// TIA Portal V20 export
FUNCTION_BLOCK "FB_Axis"   // FB410, SCL
{ S7_Optimized_Access := 'TRUE' }
// stored: AutoNumber false, MemoryReserve 100, SetENOAutomatically false
   VAR
      "sBrakeTest ZM" { S7_SetPoint := 'True'} : "FB_BrakeTest";
      "sBrakeTest ZL" { S7_SetPoint := 'True'} : "FB_BrakeTest";
      "BrakeTest ZM" : Struct
         sSBTDone { S7_SetPoint := 'True'} : Bool;
         sStartSBT { S7_SetPoint := 'True'} : Bool;
         sDone { S7_SetPoint := 'True'} : Bool;
         sError : Bool;
         sStateNum : Int;
         sDiagnoseError : Int;
         scloseExternalBrake : Bool;
      END_STRUCT;
      "BrakeTest ZL" : Struct
         sSBTDone { S7_SetPoint := 'True'} : Bool;
         sStartSBT { S7_SetPoint := 'True'} : Bool;
         sDone { S7_SetPoint := 'True'} : Bool;
         sError : Bool;
         sStateNum : Int;
         sDiagnoseError : Int;
         scloseExternalBrake : Bool;
      END_STRUCT;
      sErrorN : Array[1..8] of Bool;
      sTestStopRequested : Bool;
      sTestStopStart : Bool;
      sTestStopError : Bool;
      sTestStopEnd : Bool;
      sTestStopDone : Bool;
      sLedSITestOK : Bool;
      sLedSITestSlowFlashing : Bool;
      sLedSITestQuickFlashing : Bool;
      sTimerTestStopStart : TON_TIME;
      sTimerTestStopEnd : TON_TIME;
   END_VAR
   VAR RETAIN
      DisableAxis01_X { S7_SetPoint := 'True'} : Bool;
      DisableAxis02_Y { S7_SetPoint := 'True'} : Bool;
      DisableAxis03_ZM { S7_SetPoint := 'True'} : Bool;
      DisableAxis04_B { S7_SetPoint := 'True'} : Bool;
      DisableAxis05_U1 { S7_SetPoint := 'True'} : Bool;
      DisableAxis06_U2 { S7_SetPoint := 'True'} : Bool;
      DisableAxis07_V { S7_SetPoint := 'True'} : Bool;
      DisableAxis08_W { S7_SetPoint := 'True'} : Bool;
      DisableAxis09_ZL { S7_SetPoint := 'True'} : Bool;
   END_VAR
BEGIN
   REGION Description header 
       //==================================================================================
       // POSALUX Swiss SA / (C) Copyright 2025
       //----------------------------------------------------------------------------------
       // Title: FB_Axis
       // Comment/Function: 
       // Author: Fabien WALDT
       // Engineering: TIA Portal v17
       //----------------------------------------------------------------------------------
       // Change log table:
       // Version  | Date     | Expert in charge | Changes applied
       // ---------|----------|------------------|-----------------------------------------
       // 00.00.01 | 20250423 | WFA              | First released version
       // =================================================================================
   END_REGION

   REGION Axis disable
       "LBP_Axis01_X".A_ASpDisable  := FALSE;
       "LBP_Axis02_Y".A_ASpDisable  := FALSE;
       "LBP_Axis03_ZM".A_ASpDisable := FALSE;
       "LBP_Axis04_B".A_ASpDisable  := FALSE;
       "LBP_Axis05_U1".A_ASpDisable := FALSE;
       "LBP_Axis06_U2".A_ASpDisable := FALSE;
       "LBP_Axis07_V".A_ASpDisable  := FALSE;
       "LBP_Axis08_W".A_ASpDisable  := FALSE;
       "LBP_Axis09_ZL".A_ASpDisable := FALSE;
   END_REGION

   REGION Axis follow-up mode
       "LBP_Axis01_X".A_Follow_upMode  := TRUE;
       "LBP_Axis02_Y".A_Follow_upMode  := TRUE;
       "LBP_Axis03_ZM".A_Follow_upMode := TRUE;
       "LBP_Axis04_B".A_Follow_upMode  := TRUE;
       "LBP_Axis05_U1".A_Follow_upMode := TRUE;
       "LBP_Axis06_U2".A_Follow_upMode := TRUE;
       "LBP_Axis07_V".A_Follow_upMode  := TRUE;
       "LBP_Axis08_W".A_Follow_upMode  := TRUE;
       "LBP_Axis09_ZL".A_Follow_upMode := TRUE;
   END_REGION

   REGION Measure system selection
       "LBP_Axis01_X".A_PosMeas1  := TRUE;
       "LBP_Axis01_X".A_PosMeas2  := FALSE;
       "LBP_Axis02_Y".A_PosMeas1  := TRUE;
       "LBP_Axis02_Y".A_PosMeas2  := FALSE;
       "LBP_Axis03_ZM".A_PosMeas1 := FALSE;
       "LBP_Axis03_ZM".A_PosMeas2 := TRUE;
       "LBP_Axis04_B".A_PosMeas1  := TRUE;
       "LBP_Axis04_B".A_PosMeas2  := FALSE;
       "LBP_Axis05_U1".A_PosMeas1 := TRUE;
       "LBP_Axis05_U1".A_PosMeas2 := FALSE;
       "LBP_Axis06_U2".A_PosMeas1 := TRUE;
       "LBP_Axis06_U2".A_PosMeas2 := FALSE;
       "LBP_Axis07_V".A_PosMeas1  := TRUE;
       "LBP_Axis07_V".A_PosMeas2  := FALSE;
       "LBP_Axis08_W".A_PosMeas1  := TRUE;
       "LBP_Axis08_W".A_PosMeas2  := FALSE;
       "LBP_Axis09_ZL".A_PosMeas1 := FALSE;
       "LBP_Axis09_ZL".A_PosMeas2 := TRUE;
   END_REGION

   REGION Controle enable
       "LBP_Axis01_X".A_ContrEnable  := NOT #DisableAxis01_X;
       "LBP_Axis02_Y".A_ContrEnable  := NOT #DisableAxis02_Y;
       "LBP_Axis03_ZM".A_ContrEnable := NOT #DisableAxis03_ZM;
       "LBP_Axis04_B".A_ContrEnable  := NOT #DisableAxis04_B;
       "LBP_Axis05_U1".A_ContrEnable := NOT #DisableAxis05_U1;
       "LBP_Axis06_U2".A_ContrEnable := NOT #DisableAxis06_U2;
       "LBP_Axis07_V".A_ContrEnable  := NOT #DisableAxis07_V;
       "LBP_Axis08_W".A_ContrEnable  := NOT #DisableAxis08_W;
       "LBP_Axis09_ZL".A_ContrEnable := NOT #DisableAxis09_ZL;
   END_REGION

   REGION Pulse enable
       "LBP_Axis01_X".A_PulseEnable  := NOT #DisableAxis01_X;
       "LBP_Axis02_Y".A_PulseEnable  := NOT #DisableAxis02_Y;
       "LBP_Axis03_ZM".A_PulseEnable := NOT #DisableAxis03_ZM;
       "LBP_Axis04_B".A_PulseEnable  := NOT #DisableAxis04_B;
       "LBP_Axis05_U1".A_PulseEnable := NOT #DisableAxis05_U1;
       "LBP_Axis06_U2".A_PulseEnable := NOT #DisableAxis06_U2;
       "LBP_Axis07_V".A_PulseEnable  := NOT #DisableAxis07_V;
       "LBP_Axis08_W".A_PulseEnable  := NOT #DisableAxis08_W;
       "LBP_Axis09_ZL".A_PulseEnable := NOT #DisableAxis09_ZL;
   END_REGION

   REGION Axis04 B - Delay reference point approach
       "LBP_Axis04_B".A_DelayRef :="DB_DigitalInputs".sB_AxisReferencePoint.sSWStatus;
   END_REGION

   REGION Axis04 B - Feed Stop
       "LBP_Axis04_B".A_FDSpStop := (NOT "DB_DigitalOutputs".sClampingClosing.sSWStatus OR "DB_DigitalInputs".sClampingOpenCtrl.sSWStatus)
       OR "DB_AxisPosition".sAxis01_X."$AA_IM" < 95.0; // B Rotation diseable when X Axis is in laser area
   END_REGION

   REGION Axis05 U1 - Feed Stop
       "LBP_Axis05_U1".A_FDSpStop :=
       ("DB_LoaderShuttle1".sShuttlePosExt AND "DB_LoaderAxis".iU1PosSetPoint > "DB_AxisPosMachinePLC".Axis_U1.ExtGateExt AND NOT "DB_DigitalInputs".sExternalGateOpened.sSWStatus)       // Shuttle EXT - Consigne SAS/INT - Sas EXT pas ouvert
        OR ("DB_LoaderShuttle1".sShuttlePosSas AND "DB_LoaderAxis".iU1PosSetPoint < "DB_AxisPosMachinePLC".Axis_U1.IntGateExt AND NOT "DB_DigitalInputs".sExternalGateOpened.sSWStatus)    // Shuttle SAS - Consigne EXT     - Sas EXT pas ouvert
        OR ("DB_LoaderShuttle1".sShuttlePosSas AND "DB_LoaderAxis".iU1PosSetPoint > "DB_AxisPosMachinePLC".Axis_U1.ExtGateInt AND NOT "DB_DigitalInputs".sInternalGateOpened.sSWStatus)    // Shuttle SAS - Consigne INT     - Sas INT pas ouvert
        OR ("DB_LoaderShuttle1".sShuttlePosInt AND "DB_LoaderAxis".iU1PosSetPoint < "DB_AxisPosMachinePLC".Axis_U1.IntGateInt AND NOT "DB_DigitalInputs".sInternalGateOpened.sSWStatus)    // Shuttle INT - Consigne SAS/EXT - Sas INT pas ouvert
        OR ("DB_LoaderShuttle1".sShuttlePosInt AND NOT "DB_LoaderShuttle1".sIntLoaderInSafePos)                                                                                            // Shuttle INT - Int loader in safe position
        OR ("DB_LoaderShuttle1".sShuttlePosExt AND NOT "DB_LoaderShuttle1".sBwLoaderInSafePos) 
        OR ("DB_LoaderShuttle1".sShuttlePosExt AND "DB_BwLoader".sBwCommunication.sShuttle1Locked)
        OR ("DB_LoaderShuttle1".sShuttlePosExt AND "DB_WorkingModes".sAuto AND NOT "DB_SonplasMain".sSonplasLoader.sOutCollision);                                            // Shuttle EXT - Ext Loader in safe position
   END_REGION

   REGION Axis06 U2 - Feed Stop
       "LBP_Axis06_U2".A_FDSpStop :=
       ("DB_LoaderShuttle2".sShuttlePosExt AND "DB_LoaderAxis".iU2PosSetPoint > "DB_AxisPosMachinePLC".Axis_U2.ExtGateExt AND NOT "DB_DigitalInputs".sExternalGateOpened.sSWStatus)       // Shuttle EXT - Consigne SAS/INT - Sas EXT pas ouvert
       OR ("DB_LoaderShuttle2".sShuttlePosSas AND "DB_LoaderAxis".iU2PosSetPoint < "DB_AxisPosMachinePLC".Axis_U2.IntGateExt AND NOT "DB_DigitalInputs".sExternalGateOpened.sSWStatus)    // Shuttle SAS - Consigne EXT     - Sas EXT pas ouvert
       OR ("DB_LoaderShuttle2".sShuttlePosSas AND "DB_LoaderAxis".iU2PosSetPoint > "DB_AxisPosMachinePLC".Axis_U2.ExtGateInt AND NOT "DB_DigitalInputs".sInternalGateOpened.sSWStatus)    // Shuttle SAS - Consigne INT     - Sas INT pas ouvert
       OR ("DB_LoaderShuttle2".sShuttlePosInt AND "DB_LoaderAxis".iU2PosSetPoint < "DB_AxisPosMachinePLC".Axis_U2.IntGateInt AND NOT "DB_DigitalInputs".sInternalGateOpened.sSWStatus)    // Shuttle INT - Consigne SAS/EXT - Sas INT pas ouvert
       OR ("DB_LoaderShuttle2".sShuttlePosInt AND NOT "DB_LoaderShuttle2".sIntLoaderInSafePos)                                                                                            // Shuttle INT - Int loader in safe position 
       OR ("DB_LoaderShuttle2".sShuttlePosExt AND NOT "DB_LoaderShuttle2".sBwLoaderInSafePos)
       OR ("DB_LoaderShuttle2".sShuttlePosExt AND "DB_BwLoader".sBwCommunication.sShuttle2Locked)
       OR ("DB_LoaderShuttle2".sShuttlePosExt AND "DB_WorkingModes".sAuto AND NOT "DB_SonplasMain".sSonplasLoader.sOutCollision);                                            // Shuttle EXT - Ext Loader in safe position
   END_REGION

   REGION Axis07 V - Feed Stop
       "LBP_Axis07_V".A_FDSpStop := "DB_ExtraMissingPart".sGlobalExtraMissing;
   END_REGION

   REGION Axis08 W - Feed Stop
       "LBP_Axis08_W".A_FDSpStop := "DB_ExtraMissingPart".sGlobalExtraMissing;
   END_REGION

   REGION Check if Key Safety Stop pressed 
       IF "LBP_ModeGroup".E_JOG AND
           "DB_PowerOn".sMachinePower AND
           ("DB_McpKeyboardSignals".sK6_SITestStop.sKeySWStatus
           OR "DB_HmiKeyboardSignals".sK6_SITestStop.sKeySWStatus) THEN
           #sTestStopRequested := true;
           #sTestStopStart := false;
           #sTestStopDone := false;
           #sTestStopError := false;
       END_IF;

   END_REGION

   REGION Dynamisation forced procedure Checking (Test STOP)
       // Asking dynamisation forced
       IF #sTestStopRequested THEN
           IF ("LBP_Axis01_X".SIC.SW2.TestStopReq OR 
               "LBP_Axis02_Y".SIC.SW2.TestStopReq OR
               "LBP_Axis03_ZM".SIC.SW2.TestStopReq OR
               "LBP_Axis04_B".SIC.SW2.TestStopReq OR
               "LBP_Axis05_U1".SIC.SW2.TestStopReq OR
               "LBP_Axis06_U2".SIC.SW2.TestStopReq OR
               "LBP_Axis07_V".SIC.SW2.TestStopReq OR
               "LBP_Axis08_W".SIC.SW2.TestStopReq OR
               "LBP_Axis09_ZL".SIC.SW2.TestStopReq)
           THEN
               "LBP_Axis01_X".SCC.CW1.TeststopStart := TRUE; 
               "LBP_Axis02_Y".SCC.CW1.TeststopStart := TRUE;
               "LBP_Axis03_ZM".SCC.CW1.TeststopStart := TRUE;
               "LBP_Axis04_B".SCC.CW1.TeststopStart := TRUE;
               "LBP_Axis05_U1".SCC.CW1.TeststopStart := TRUE;
               "LBP_Axis06_U2".SCC.CW1.TeststopStart := TRUE;
               "LBP_Axis07_V".SCC.CW1.TeststopStart := TRUE;
               "LBP_Axis08_W".SCC.CW1.TeststopStart := TRUE;
               "LBP_Axis09_ZL".SCC.CW1.TeststopStart := TRUE;
               #sTestStopStart := TRUE;
           ELSE
               #sTestStopDone := TRUE;
               #"BrakeTest ZM".sStartSBT := TRUE;
               #"BrakeTest ZM".sSBTDone := FALSE;
               #"BrakeTest ZL".sStartSBT := TRUE;
               #"BrakeTest ZL".sSBTDone := FALSE;
           END_IF;
           #sTestStopRequested := FALSE;
       END_IF;

       //Timer dynamisation forced : Begin 
       #sTimerTestStopStart.TON (IN := #sTestStopStart,
       PT := t#500ms);

       //Reset dynamisation forcée
       IF #sTimerTestStopStart.Q THEN
           IF "LBP_Axis01_X".SIC.SW2.TestStopAct AND 
               "LBP_Axis02_Y".SIC.SW2.TestStopAct AND
               "LBP_Axis03_ZM".SIC.SW2.TestStopAct AND
               "LBP_Axis04_B".SIC.SW2.TestStopAct AND
               "LBP_Axis05_U1".SIC.SW2.TestStopAct AND
               "LBP_Axis06_U2".SIC.SW2.TestStopAct AND
               "LBP_Axis07_V".SIC.SW2.TestStopAct AND
               "LBP_Axis08_W".SIC.SW2.TestStopAct AND
               "LBP_Axis09_ZL".SIC.SW2.TestStopAct 
           THEN
               "LBP_Axis01_X".SCC.CW1.TeststopStart := FALSE;
               "LBP_Axis02_Y".SCC.CW1.TeststopStart := FALSE;
               "LBP_Axis03_ZM".SCC.CW1.TeststopStart := FALSE;
               "LBP_Axis04_B".SCC.CW1.TeststopStart := FALSE;
               "LBP_Axis05_U1".SCC.CW1.TeststopStart := FALSE;
               "LBP_Axis06_U2".SCC.CW1.TeststopStart := FALSE;
               "LBP_Axis07_V".SCC.CW1.TeststopStart := FALSE;
               "LBP_Axis08_W".SCC.CW1.TeststopStart := FALSE;
               "LBP_Axis09_ZL".SCC.CW1.TeststopStart := FALSE;

               #sTestStopEnd := TRUE;
               #sTestStopStart := FALSE;
           END_IF;
       END_IF;

       //Timer dynamisation forced : End 
       #sTimerTestStopEnd.TON (IN := #sTestStopEnd,
       PT := t#500ms);

       IF #sTimerTestStopEnd.Q THEN

           IF "LBP_Axis01_X".SIC.SW2.TestStopReq         
               OR "LBP_Axis02_Y".SIC.SW2.TestStopReq
               OR "LBP_Axis03_ZM".SIC.SW2.TestStopReq
               OR "LBP_Axis04_B".SIC.SW2.TestStopReq
               OR "LBP_Axis05_U1".SIC.SW2.TestStopReq
               OR "LBP_Axis06_U2".SIC.SW2.TestStopReq
               OR "LBP_Axis07_V".SIC.SW2.TestStopReq
               OR "LBP_Axis08_W".SIC.SW2.TestStopReq
               OR "LBP_Axis09_ZL".SIC.SW2.TestStopReq
           THEN
               #sTestStopError := TRUE;
           END_IF;
           #sTestStopEnd := FALSE;
           #sTestStopDone := TRUE;

           #"BrakeTest ZM".sStartSBT := TRUE;
           #"BrakeTest ZM".sSBTDone := FALSE;
           #"BrakeTest ZL".sStartSBT := TRUE;
           #"BrakeTest ZL".sSBTDone := FALSE;
       END_IF;

       "LBP_AlarmMsgs".UserA[5].A70UUxx[43] := #sTestStopError;  // Msg 700543 : SAFETY: TEST STOP ERROR

       IF "MCP1_In".reset THEN
           "LBP_Axis01_X".SCC.CW1.TeststopStart := FALSE; 
           "LBP_Axis02_Y".SCC.CW1.TeststopStart := FALSE;
           "LBP_Axis03_ZM".SCC.CW1.TeststopStart := FALSE;
           "LBP_Axis04_B".SCC.CW1.TeststopStart := FALSE;
           "LBP_Axis05_U1".SCC.CW1.TeststopStart := FALSE;
           "LBP_Axis06_U2".SCC.CW1.TeststopStart := FALSE;
           "LBP_Axis07_V".SCC.CW1.TeststopStart := FALSE;
           "LBP_Axis08_W".SCC.CW1.TeststopStart := FALSE;
           "LBP_Axis09_ZL".SCC.CW1.TeststopStart := FALSE;

           #sTestStopRequested := FALSE;
           #sTestStopStart := FALSE;
       END_IF;
   END_REGION

   REGION Safe Brake Test Control (SBT) - Z axis

       IF "MCP1_In".reset OR NOT "LBP_ModeGroup".E_JOG THEN
           #"BrakeTest ZM".sStartSBT := FALSE;
           #"BrakeTest ZL".sStartSBT := FALSE;
       END_IF;

       #"sBrakeTest ZM"(iStartBt := #"BrakeTest ZM".sStartSBT,
                   iQuit := "MCP1_In".reset,
                   iExternalBrakeClosed := false,
                   iMaxStepTime := T#10S,
                   iBrakeNum := false,
                   iActivateAutoDirection := false,
                   iSetManualDirection := false,
                   iTestSequence := false,
                   oCloseExternalBrake => #"BrakeTest ZM".scloseExternalBrake,
                   oDone => #"BrakeTest ZM".sDone,
                   oError => #"BrakeTest ZM".sError,
                   oStateNum => #"BrakeTest ZM".sStateNum,
                   oDiagnoseError => #"BrakeTest ZM".sDiagnoseError,
                   oError1 => #sErrorN[1],
                   oError2 => #sErrorN[2],
                   oError3 => #sErrorN[3],
                   oError4 => #sErrorN[4],
                   oError5 => #sErrorN[5],
                   oError6 => #sErrorN[6],
                   oError7 => #sErrorN[7],
                   oError8 => #sErrorN[8],
                   ioAxisDB := "LBP_Axis03_ZM");

   #"sBrakeTest ZL"(iStartBt := #"BrakeTest ZL".sStartSBT,
                     iQuit := "MCP1_In".reset,
                     iExternalBrakeClosed := false,
                     iMaxStepTime := T#10S,
                     iBrakeNum := false,
                     iActivateAutoDirection := false,
                     iSetManualDirection := false,
                     iTestSequence := false,
                     oCloseExternalBrake => #"BrakeTest ZL".scloseExternalBrake,
                     oDone => #"BrakeTest ZL".sDone,
                     oError => #"BrakeTest ZL".sError,
                     oStateNum => #"BrakeTest ZL".sStateNum,
                     oDiagnoseError => #"BrakeTest ZL".sDiagnoseError,
                     oError1 => #sErrorN[1],
                     oError2 => #sErrorN[2],
                     oError3 => #sErrorN[3],
                     oError4 => #sErrorN[4],
                     oError5 => #sErrorN[5],
                     oError6 => #sErrorN[6],
                     oError7 => #sErrorN[7],
                     oError8 => #sErrorN[8],
                     ioAxisDB := "LBP_Axis09_ZL");

    IF #"BrakeTest ZM".sDone AND #"BrakeTest ZL".sDone THEN
        #"BrakeTest ZM".sStartSBT := FALSE;
        #"BrakeTest ZM".sSBTDone := TRUE;
        #"BrakeTest ZL".sStartSBT := FALSE;
        #"BrakeTest ZL".sSBTDone := TRUE;
           "LBP_AlarmMsgs".UserA[5].A70UUxx[12] := FALSE;  // Msg 700512 "SAFETY: THE BRAKE TEST IS NOT WORKING, PLEASE RESET"
       END_IF;

       IF #"BrakeTest ZM".sDiagnoseError <> 0 AND #"BrakeTest ZL".sDiagnoseError <> 0 THEN
           "LBP_AlarmMsgs".UserA[5].A70UUxx[12] := TRUE;  // Msg 700512 "SAFETY: THE BRAKE TEST IS NOT WORKING, PLEASE RESET"
       END_IF;

   END_REGION

   REGION LED SAFETY TEST 
       #sLedSITestSlowFlashing :=
       "LBP_ModeGroup".E_JOG
       AND "DB_PowerOn".sMachinePower
       AND NOT #"BrakeTest ZM".sStartSBT
       AND NOT #"BrakeTest ZL".sStartSBT
       AND NOT #sTestStopStart
       AND "DB_DataFromSafety".DoorsClosed
       AND (NOT #"BrakeTest ZM".sSBTDone
           OR NOT #"BrakeTest ZL".sSBTDone
           OR NOT #sTestStopDone
           OR "LBP_Axis01_X".SIC.SW2.TestStopReq     
           OR "LBP_Axis02_Y".SIC.SW2.TestStopReq
           OR "LBP_Axis03_ZM".SIC.SW2.TestStopReq
           OR "LBP_Axis04_B".SIC.SW2.TestStopReq
           OR "LBP_Axis05_U1".SIC.SW2.TestStopReq
           OR "LBP_Axis06_U2".SIC.SW2.TestStopReq
           OR "LBP_Axis07_V".SIC.SW2.TestStopReq
           OR "LBP_Axis08_W".SIC.SW2.TestStopReq
           OR "LBP_Axis09_ZL".SIC.SW2.TestStopReq);
       #sLedSITestQuickFlashing :=
       ("LBP_AlarmMsgs".UserA[5].A70UUxx[12]              // Msg 700512 "SAFETY: THE BRAKE TEST IS NOT WORKING, PLEASE RESET"
           OR "LBP_AlarmMsgs".UserA[5].A70UUxx[43])       // Msg 700543 "SAFETY: TEST STOP ERROR"
           AND "DB_PowerOn".sMachinePower;

       #sLedSITestOK :=
       NOT #"BrakeTest ZM".sStartSBT
           AND NOT  #"BrakeTest ZL".sStartSBT
           AND NOT #sTestStopStart
           AND NOT "LBP_AlarmMsgs".UserA[5].A70UUxx[12]   // Msg 700512 "SAFETY: THE BRAKE TEST IS NOT WORKING, PLEASE RESET"
           AND NOT "LBP_AlarmMsgs".UserA[5].A70UUxx[43]   // Msg 700543 "SAFETY: TEST STOP ERROR"
           AND #"BrakeTest ZM".sSBTDone
           AND #"BrakeTest ZL".sSBTDone
           AND #sTestStopDone
           AND NOT #sLedSITestSlowFlashing
           AND NOT #sLedSITestQuickFlashing;

           "DB_McpKeyboardSignals".sK6_SITestStop.sLedSWStatus :=     
           #sLedSITestOK
           OR (#sLedSITestSlowFlashing AND "Clock_1Hz")
           OR (#sLedSITestQuickFlashing AND "Clock_2Hz");

           "DB_HmiKeyboardSignals".sK6_SITestStop.sLedSWStatus :=
           #sLedSITestOK
           OR (#sLedSITestSlowFlashing AND "Clock_1Hz")
           OR (#sLedSITestQuickFlashing AND "Clock_2Hz");
   END_REGION
END_FUNCTION_BLOCK
